// TIA Portal V20 export
FUNCTION_BLOCK "Conveyor_C3"   // FB10026, FBD
// stored: Access Published, MemoryReserve 100, Namespace C3, SetENOAutomatically false
   VAR
      R_TRIG_Instance { S7_SetPoint := 'True'} : R_TRIG;
      StatAutoRight { S7_SetPoint := 'True'} : Bool;
   END_VAR
BEGIN

REGION Network 1: Run conveyor LEFT
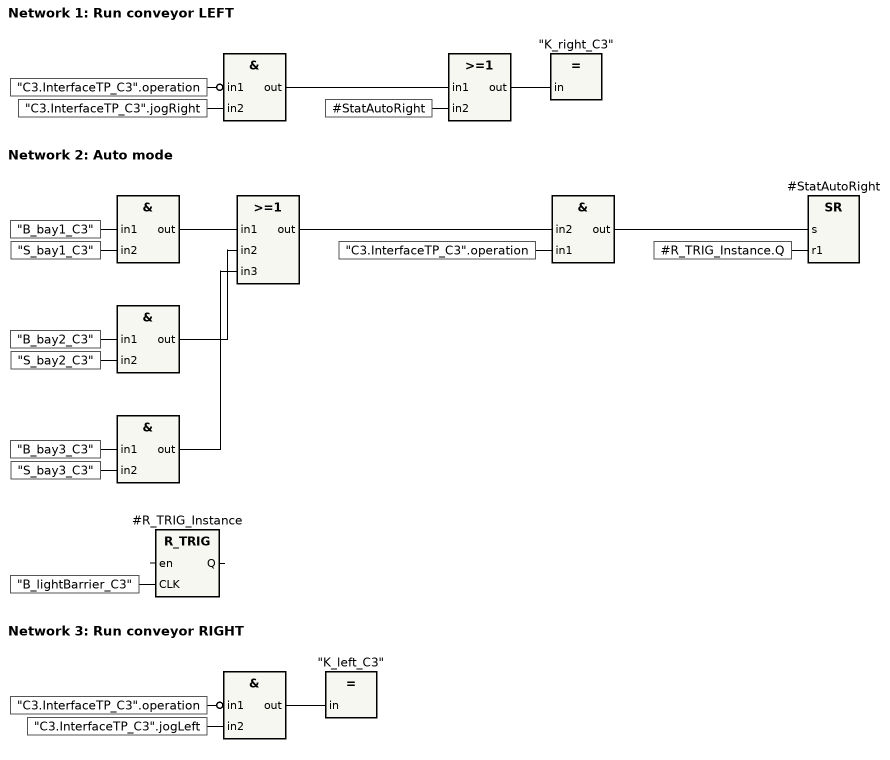
   "K_right_C3" := (NOT "C3.InterfaceTP_C3".operation AND "C3.InterfaceTP_C3".jogRight) OR #StatAutoRight;
END_REGION

REGION Network 2: Auto mode
   IF (("B_bay1_C3" AND "S_bay1_C3") OR ("B_bay2_C3" AND "S_bay2_C3") OR ("B_bay3_C3" AND "S_bay3_C3")) AND "C3.InterfaceTP_C3".operation THEN
       #StatAutoRight := TRUE;   // SR flip-flop
   END_IF;
   IF #R_TRIG_Instance.Q THEN #StatAutoRight := FALSE; END_IF;
   #R_TRIG_Instance(CLK := "B_lightBarrier_C3");   // R_TRIG
END_REGION

REGION Network 3: Run conveyor RIGHT
   "K_left_C3" := NOT "C3.InterfaceTP_C3".operation AND "C3.InterfaceTP_C3".jogLeft;
END_REGION
END_FUNCTION_BLOCK
